INTERFACE I_Nci_Ctrl

PROPERTY ChnId : udint
GET
END_GET
END_PROPERTY

METHOD Cycle
VAR_INPUT
END_VAR
END_METHOD

PROPERTY eCmd : E_NCI_CTRL
GET
END_GET
SET
END_SET
END_PROPERTY

PROPERTY eState : E_NCI_CTRL
GET
END_GET
SET
END_SET
END_PROPERTY

PROPERTY GroupAxisConfig : ST_3D_Group
GET
END_GET
SET
END_SET
END_PROPERTY

PROPERTY I_AuxAxis : array[1..GVL_NCI.cAuxAxisCount] of I_McAxis
GET
END_GET
SET
END_SET
END_PROPERTY

PROPERTY I_McAxis : array[1..GVL_NCI.cMcAxisCount] of I_McAxis
GET
END_GET
SET
END_SET
END_PROPERTY

PROPERTY I_NcChannel : I_NciChannel
GET
END_GET
END_PROPERTY

PROPERTY M_FuncReq : word
GET
END_GET
END_PROPERTY

PROPERTY NcProg : string(255)
GET
END_GET
SET
END_SET
END_PROPERTY

PROPERTY R_Param_Read : ARRAY [0..GVL_NCI.cRParamCount] OF lreal
GET
END_GET
SET
END_SET
END_PROPERTY

PROPERTY R_Param_Write : ARRAY [0..GVL_NCI.cRParamCount] OF lreal
GET
END_GET
SET
END_SET
END_PROPERTY

PROPERTY R_ParamCount : DINT
GET
END_GET
SET
END_SET
END_PROPERTY

PROPERTY R_ParamIndex : DINT
GET
END_GET
SET
END_SET
END_PROPERTY

PROPERTY sCmd : string
GET
END_GET
SET
END_SET
END_PROPERTY

END_INTERFACE

(* stored: Version 1.1.0.1, ProductVersion 3.1.4024.12
   Itf I_Nci_Ctrl: Id {07cae18a-edd8-0c79-0290-3533a7fb6aa9}
   Folder methods: Id {f1063346-b567-0cec-37b4-73f99aec2ce1}
   Folder properties: Id {3965fb1f-36ec-04ff-058c-946b7a8d2d04}
   Property ChnId: Id {550574a7-3465-07d8-3e15-1fa15c6d0b67}
   Get Get: Id {23c2b759-bad2-065e-2a33-1cb335cd8792}
   Method Cycle: Id {05ec7737-5f93-0b30-38ee-c896f70763b2}
   Property eCmd: Id {82dec9b9-63d6-0bd1-184b-ce3d10fff674}
   Get Get: Id {c41f9e03-bf25-0f54-39fb-9d5004ad695a}
   Set Set: Id {8d0ec2ba-2ecc-0384-2c89-c91395ba9494}
   Property eState: Id {6593e121-53e8-0f2f-24af-2d5172c41b34}
   Get Get: Id {d19232bf-e53b-0e9a-21ba-a170037c4d97}
   Set Set: Id {81a59c9b-1133-0b6d-2675-dd5939dce4d4}
   Property GroupAxisConfig: Id {2258ed59-a296-07fd-389e-c9db1a3ae19d}
   Get Get: Id {76b98d0f-1d76-05da-11cd-f6a6a5d1eeee}
   Set Set: Id {eb622bec-68da-0f65-0ed3-91978a4565c8}
   Property I_AuxAxis: Id {f6b970a6-97dc-0826-3c41-44b34500e9e4}
   Get Get: Id {cc7dbf2a-d9f3-006e-3c13-36101b958cdc}
   Set Set: Id {7a03f9b9-9604-0003-08ac-4993e168cab4}
   Property I_McAxis: Id {b79ec8b1-aef9-072a-362d-afc0cb0a65a4}
   Get Get: Id {7bcb28a3-c371-0118-1eb8-efe57aec73cf}
   Set Set: Id {738e5654-8107-09f4-0685-4112ae5e925d}
   Property I_NcChannel: Id {31caac85-480c-052e-0d15-358e52677b2f}
   Get Get: Id {80a20f2c-d2ef-0196-317b-2fce68b126a9}
   Property M_FuncReq: Id {c6bf003d-18f0-01c1-3d1d-8aaa286da1d1}
   Get Get: Id {53e26ef5-94dc-0681-1449-e3b9be0bb0ea}
   Property NcProg: Id {84919416-a902-0453-3db9-63c707919993}
   Get Get: Id {38154da0-5475-0fbb-2ea4-6285efe52f0b}
   Set Set: Id {71cc54d2-739a-052b-3f03-03bcc215a1ec}
   Property R_Param_Read: Id {b1108182-3b32-0621-0899-25029c9dae74}
   Get Get: Id {3aca5d0f-5898-0793-03e4-8175e7d47b80}
   Set Set: Id {559e5a94-181a-070b-1200-8d71b07ed055}
   Property R_Param_Write: Id {57e12b4b-7ae9-0dd6-3f69-4b7a38207a88}
   Get Get: Id {57a210db-09d7-010e-0104-694af83d11cf}
   Set Set: Id {41b9dc1e-2c50-0bb7-0447-ed07da198877}
   Property R_ParamCount: Id {556c6da9-54f7-0f69-14c3-6e12d8af1c9f}
   Get Get: Id {479dae77-8644-0e7a-124b-2b1cc2562772}
   Set Set: Id {9fd4fd70-e9f8-0142-2d5a-cf13cf4fd1e4}
   Property R_ParamIndex: Id {6dd144d3-e54b-08d0-147a-9e984ed8498e}
   Get Get: Id {97ff0744-c9f0-0f1e-2f30-55dc436f2323}
   Set Set: Id {c820f92e-d200-0bfc-270c-64bee9ccda7e}
   Property sCmd: Id {1da1638c-b9ab-0271-0d67-3215818fd514}
   Get Get: Id {c97f8e35-07d0-0a0a-2f19-320336098439}
   Set Set: Id {f9287450-b674-0d9b-057f-1bece409bc05} *)
